FUNCTION_BLOCK E_F_TRIG (* Boolean falling edge detection *)
  (* Standard: 61499-1; Classification: Event handling; Function: Edge detection *)
  (* Version 0.1, 2002-01-29, JHC, Rockwell Automation, XML version *)
  (* Version 0.0, 1998-10-12, JHC, Rockwell Automation, SRC version *)
  (* Compiler header: package fb.rt.events; *)
  (* Compiler Java IBM VisualAge 3.0 *)
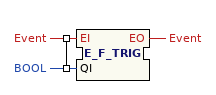
  EVENT_INPUT
    EI WITH QI; (* Event Input *)
  END_EVENT
  EVENT_OUTPUT
    EO; (* Event Output *)
  END_EVENT
  VAR_INPUT
    QI : BOOL; (* Boolean input for falling edge detection *)
  END_VAR
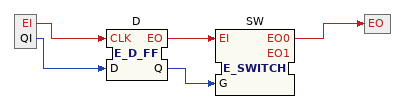
  FBS
    D : E_D_FF;
    SW : E_SWITCH;
  END_FBS
  EVENT_CONNECTIONS
    EI TO D.CLK;
    D.EO TO SW.EI;
    SW.EO0 TO EO;
  END_CONNECTIONS
  DATA_CONNECTIONS
    QI TO D.D;
    D.Q TO SW.G;
  END_CONNECTIONS
END_FUNCTION_BLOCK
